# EPICS substitutions: db/Beckhoff_3XXX/ecmcEL3356.substitutions
file "ecmc_analogInput-chX.template"
{
  pattern { CH_ID,  ESLO,  EGU,    PREC }
          { 01,     1.0,   "RAW",  3 }
}

file "ecmc_status_analog-chX.template"
{
  pattern {CH_ID, KEY }
          {01,    "AI"}
}
